ABB RAPID module: Module2023_simulada.mod

MODULE Module1
	CONST robtarget Pos_origen:=[[495,-250,560],[0,0,1,0],[-1,-1,-1,0],[9E+09,9E+09,9E+09,9E+09,9E+09,9E+09]];
	CONST robtarget Pos_prepick_Brick:=[[486,-578,484],[0,0,1,0],[-1,-1,-2,0],[9E+09,9E+09,9E+09,9E+09,9E+09,9E+09]];
	CONST robtarget Pos_pick_Brick:=[[486,-578,404],[0,0,1,0],[-1,-1,-2,0],[9E+09,9E+09,9E+09,9E+09,9E+09,9E+09]];
	CONST robtarget Pos_preplace_Brick:=[[610,-230,345],[0,0,1,0],[-1,-1,-1,0],[9E+09,9E+09,9E+09,9E+09,9E+09,9E+09]];
	CONST robtarget Pos_place_Brick:=[[610,-230,265.7],[0,0,1,0],[-1,-1,-1,0],[9E+09,9E+09,9E+09,9E+09,9E+09,9E+09]];
	CONST robtarget Pos_prepick_lata:=[[427,-575,491],[0,0,1,0],[-1,-1,-2,0],[9E+09,9E+09,9E+09,9E+09,9E+09,9E+09]];
	CONST robtarget Pos_pick_lata:=[[427,-575,411],[0,0,1,0],[-1,-1,-2,0],[9E+09,9E+09,9E+09,9E+09,9E+09,9E+09]];
	CONST robtarget Pos_preplace_lata:=[[587,26,360],[0,0,1,0],[0,-1,-1,0],[9E+09,9E+09,9E+09,9E+09,9E+09,9E+09]];
	CONST robtarget Pos_place_lata:=[[587,26,280],[0,0,1,0],[0,-1,-1,0],[9E+09,9E+09,9E+09,9E+09,9E+09,9E+09]];
    VAR robtarget prepick_var;
    VAR robtarget pick_var;
ENDMODULE
